{attribute 'GeneratedUsingTerminal: EK1960-2600-0019'}
{attribute addProperty BoxType "EK1960-2600-0019"}
{attribute addProperty Id "FSoE_InputsFSoE_Inputs_905C193448FSoE_OutputsFSoE_Outputs_77F9785A56"}
{attribute addProperty CRC "2121031902"}
{attribute addProperty Size "104"}
TYPE Module_1_FSoE_7E6C60DE :
STRUCT
	{attribute addProperty Name "FSoE_Inputs"}
	FSoE_Inputs  : FSoE_Inputs_905C1934;
	{attribute addProperty Name "FSoE_Outputs"}
	FSoE_Outputs  : FSoE_Outputs_77F9785A;
END_STRUCT
END_TYPE

(* stored: Version 1.2.0.0, ProductVersion 3.1.4024.11
   DUT Module_1_FSoE_7E6C60DE: Id {8478df5f-13b7-4f9b-9e86-b493d475315b} *)
